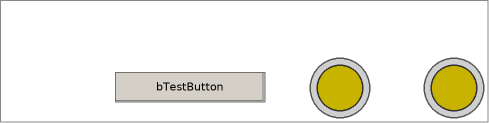
VISUALIZATION VISU_Simulation  // 489x123
    Button (115,72 150x30), "bTestButton"
        tap MAIN.fbSimulationInputs.bDummyRoomButton
    Lamp1 (305,53 70x70), variable: MAIN.fbSimulationOutputs.bDummyRoomLight1Relay, style: Lamp-Lamp1-Yellow
    Lamp1 (419,53 70x70), variable: MAIN.fbSimulationOutputs.bDummyRoomLight2Relay, style: Lamp-Lamp1-Yellow
END_VISUALIZATION

(* stored: Version 1.1.0.1
   Visu VISU_Simulation: Id {181cc198-ebd5-4598-9e66-87cb1548e48a} *)
